(* CoDeSys 2.3.9.42 project: CANOPEN_ROBOTEQ_DRAAIENDE_MOTOR.pro *)
(* Libraries: ifm_CANopen\ifm_CANopen_NT_V020004.lib 3.11.15 18:07:50, SysLibPlcCtrl.lib 13.6.03 15:49:00, SysLibFile.lib 23.9.04 10:11:36, SysLibTime.lib 27.4.05 10:36:52, SysLibTargetVisu.lib 5.4.04 13:31:00, LinuxSystemLib.Lib 18.3.03 12:26:50, ifm_pdm_file_V010006.lib 14.1.08 13:21:32, ifm_CR0403\ifm_CR0403_V030100.lib 15.1.16 14:49:16, ifm_J1939_NT\ifm_J1939_NT_V020004.lib 18.9.14 16:13:02, ifm_RAWCan\ifm_RAWCan_NT_V020004.lib 3.11.15 18:07:52, standard.lib 4.10.05 11:14:46, SysLibCallback.lib 26.9.08 17:43:52, Util.lib 6.11.07 15:39:24 *)

(* PLC configuration (modules and I/O channels)
Configuration [LocalConfiguration] node 0, in %IB0 out %QB0 {IFM_PARAM_WORD_TIME = 0}
Inputs Binary [LocalIn] node 0, in %IB0 out %QB0
  IN00 AT %IB0 [ChInputBool] Input 00 Bit
  IN01 AT %IB1 [ChInputBool] Input 01 Bit
  IN02 AT %IB2 [ChInputBool] Input 02 Bit
  IN03 AT %IB3 [ChInputBool] Input 03 Bit
  IN04 AT %IB4 [ChInputBool] Input 04 Bit
  IN05 AT %IB5 [ChInputBool] Input 05 Bit
  IN06 AT %IB6 [ChInputBool] Input 06 Bit
  IN07 AT %IB7 [ChInputBool] Input 07 Bit
  IN08 AT %IB8 [ChInputBool] Input 08 Bit
  IN09 AT %IB9 [ChInputBool] Input 09 Bit
  IN10 AT %IB10 [ChInputBool] Input 10 Bit
  IN11 AT %IB11 [ChInputBool] Input 11 Bit
Outputs Binary [LocalOut] node 1, in %IB12 out %QB0
  OUT00 AT %QB0 [ChOutputBool] Output 00 Bit
  OUT01 AT %QB1 [ChOutputBool] Output 01 Bit
  OUT02 AT %QB2 [ChOutputBool] Output 02 Bit
  OUT03 AT %QB3 [ChOutputBool] Output 03 Bit
  OUT04 AT %QB4 [ChOutputBool] Output 04 Bit
  OUT05 AT %QB5 [ChOutputBool] Output 05 Bit
  OUT06 AT %QB6 [ChOutputBool] Output 06 Bit
  OUT07 AT %QB7 [ChOutputBool] Output 07 Bit
  OUT08 AT %QB8 [ChOutputBool] Output 08 Bit
  OUT09 AT %QB9 [ChOutputBool] Output 09 Bit
  OUT10 AT %QB10 [ChOutputBool] Output 10 Bit
  OUT11 AT %QB11 [ChOutputBool] Output 11 Bit
System Inputs [LocalSystemInputs] node 2, in %IB12 out %QB12
  SUPPLY_VOLTAGE_VBBS AT %IW6 [ChInputWord] Supply voltage VBBS
  SUPPLY_VOLTAGE_VU AT %IW7 [ChInputWord] Supply voltage VU
  SUPPLY_VOLTAGE_VBB1 AT %IW8 [ChInputWord] Supply voltage VBB1
  SUPPLY_VOLTAGE_VBB2 AT %IW9 [ChInputWord] Supply voltage VBB2
  TEMPERATURE AT %IW10 [ChInputInt] Temperature
J1939 Interface [CAN_J1939] node 1, in %IB56 out %QB44
CANopen Master [CanMaster] node 0, in %IB56 out %QB44
J1939 Interface [CAN_J1939] node 1, in %IB56 out %QB44
*)

(* POU PLC_PRG, ST *)
PROGRAM PLC_PRG
VAR

	CAN_ENABLE_CH2_125: CAN_ENABLE;
	CAN_ENABLE_CH1_125: CAN_ENABLE;

END_VAR
CAN_ENABLE_CH1_125(ENABLE:=TRUE , CHANNEL:=1 , BAUDRATE:=125 , RESULT=> );

CAN_ENABLE_CH2_125(ENABLE:=TRUE , CHANNEL:=2 , BAUDRATE:=250 , RESULT=> );

(*
Velocity1:=1000;
Velocity2:=1000;
*)
(*
CANOPEN_SDOWRITE_(
	EXECUTE:= , 
	CHANNEL:= , 
	NODE:= , 
	IDX:= , 
	SUBIDX:= , 
	LEN:= , 
	DATA:= , 
	Timeout:= , 
	RESULT=> );
*)
END_PROGRAM

(* Visualisation roboteq
2 more shapes without text or variables
*)
